FUNCTION_BLOCK FB_ThNTZ_Stellwertscheck
VAR_IN_OUT
	Stellwert	: ST_ThNTZ_Stellwert;
END_VAR

VAR_INPUT
	Parameter	: ST_ThNTZ_Parameter;
END_VAR
VAR_OUTPUT
END_VAR
VAR
END_VAR

IF( Stellwert.Betrieb ) THEN
	(* Max-Min-Grenzen erzwingen *)
	Stellwert.Leistung		 := MIN(Parameter.Stellwert_Leistung_max, Stellwert.Leistung);
	Stellwert.Leistung		 := MAX(Parameter.Stellwert_Leistung_min, Stellwert.Leistung);
ELSE
	Stellwert.Leistung		 := 0;
END_IF;

END_FUNCTION_BLOCK

(* stored: Version 1.1.0.1, ProductVersion 3.1.4024.9
   POU FB_ThNTZ_Stellwertscheck: Id {748f8609-7fa1-4185-b9a2-4ac31678fd4e}, SpecialFunc None *)
